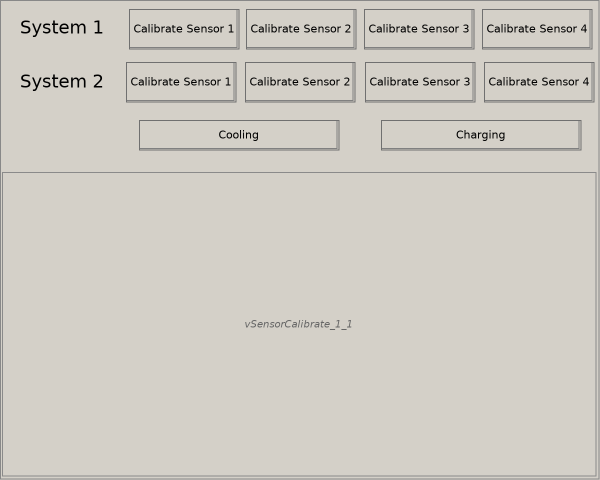
VISUALIZATION vCalibrationScreen  // 600x480
    Button (129,9 110x40), "Calibrate Sensor 1"
        OnMouseClick: FrameSelectionChange Selection=SelectedFrame=5ae10b84-1184-4faf-a213-c28aed3d2f26, GlobSel=AssignType=Directly, SelType=Locally
    Button (246,9 110x40), "Calibrate Sensor 2"
        OnMouseClick: FrameSelectionChange Selection=SelectedFrame=5ae10b84-1184-4faf-a213-c28aed3d2f26, Selection=1, GlobSel=AssignType=Directly, SelType=Locally
    Label (8,15 108x25), "System 1"
    Button (364,9 110x40), "Calibrate Sensor 3"
        OnMouseClick: FrameSelectionChange Selection=SelectedFrame=5ae10b84-1184-4faf-a213-c28aed3d2f26, Selection=2, GlobSel=AssignType=Directly, SelType=Locally
    Button (482,9 110x40), "Calibrate Sensor 4"
        OnMouseClick: FrameSelectionChange Selection=SelectedFrame=5ae10b84-1184-4faf-a213-c28aed3d2f26, Selection=3, GlobSel=AssignType=Directly, SelType=Locally
    Button (126,62 110x40), "Calibrate Sensor 1"
        OnMouseClick: FrameSelectionChange Selection=SelectedFrame=5ae10b84-1184-4faf-a213-c28aed3d2f26, Selection=4, GlobSel=AssignType=Directly, SelType=Locally
    Button (245,62 110x40), "Calibrate Sensor 2"
        OnMouseClick: FrameSelectionChange Selection=SelectedFrame=5ae10b84-1184-4faf-a213-c28aed3d2f26, Selection=5, GlobSel=AssignType=Directly, SelType=Locally
    Label (8,69 108x25), "System 2"
    Button (365,62 110x40), "Calibrate Sensor 3"
        OnMouseClick: FrameSelectionChange Selection=SelectedFrame=5ae10b84-1184-4faf-a213-c28aed3d2f26, Selection=6, GlobSel=AssignType=Directly, SelType=Locally
    Button (484,62 110x40), "Calibrate Sensor 4"
        OnMouseClick: FrameSelectionChange Selection=SelectedFrame=5ae10b84-1184-4faf-a213-c28aed3d2f26, Selection=7, GlobSel=AssignType=Directly, SelType=Locally
    Frame (2,172 594x304)
        shows vSensorCalibrate_1_1(vAnalogSensor := ACTION1.fbAnalogSensor1)
        shows vSensorCalibrate_1_2(vAnalogSensor := ACTION1.fbAnalogSensor2)
        shows vSensorCalibrate_1_3(vAnalogSensor := ACTION1.fbAnalogSensor3)
        shows vSensorCalibrate_1_4(vAnalogSensor := ACTION1.fbAnalogSensor4)
        shows vSensorCalibrate_2_1(vAnalogSensor := ACTION2.fbAnalogSensor1)
        shows vSensorCalibrate_2_2(vAnalogSensor := ACTION2.fbAnalogSensor2)
        shows vSensorCalibrate_2_3(vAnalogSensor := ACTION2.fbAnalogSensor3)
        shows vSensorCalibrate_2_4(vAnalogSensor := ACTION2.fbAnalogSensor4)
        shows vCharging()
        shows vCooling()
    Button (139,120 200x30), "Cooling"
        OnMouseClick: FrameSelectionChange Selection=SelectedFrame=5ae10b84-1184-4faf-a213-c28aed3d2f26, Selection=9, GlobSel=AssignType=Directly, SelType=Locally
    Button (381,120 200x30), "Charging"
        OnMouseClick: FrameSelectionChange Selection=SelectedFrame=5ae10b84-1184-4faf-a213-c28aed3d2f26, Selection=8, GlobSel=AssignType=Directly, SelType=Locally
END_VISUALIZATION

(* stored: Version 1.1.0.1, ProductVersion 3.1.4024.12
   Visu vCalibrationScreen: Id {ea46625d-7295-48f9-a566-23da2abf9846} *)
